Staubli VAL3: sendAckIO.pgx

public program sendAckIO(sio& x_sSocket, num& x_nConnFlag, RosSimpleMsg& x_rMsg, num& x_nMsgRecvState)
begin
  // Copyright (c) 2016, Ocado Technology - Robotics Research Team
  //
  // Licensed under the Apache License, Version 2.0 (the "License");
  // you may not use this file except in compliance with the License.
  // You may obtain a copy of the License at
  //
  //     http://www.apache.org/licenses/LICENSE-2.0
  //
  // Unless required by applicable law or agreed to in writing, software
  // distributed under the License is distributed on an "AS IS" BASIS,
  // WITHOUT WARRANTIES OR CONDITIONS OF ANY KIND, either express or implied.
  // See the License for the specific language governing permissions and
  // limitations under the License.



  switch x_rMsg.header.nMsgType
    case nStdMsgType["JOINT_TRAJ_PT"]
      call sendRosMsg(siTcpIpMotion, rosTrajPtAck.prefix, rosTrajPtAck.header, rosTrajPtAck.body, nInConnFlag)
    break
    case nStdMsgType["JOINT_TRAJ_PT_FULL"]
      call sendRosMsg(siTcpIpMotion, rosTrajPtFAck.prefix, rosTrajPtFAck.header, rosTrajPtFAck.body, nInConnFlag)
    break
    case Staubli:MsgType.WRITE_SINGLE_IO
      call sendRosMsg(x_sSocket, Staubli:writeSingIOAck.prefix, Staubli:writeSingIOAck.header, Staubli:writeSingIOAck.body, x_nConnFlag)
    break
    default
    break
  endSwitch

  // regardless of result from sending ACK
  // reset state machine to receive new messages
  x_nMsgRecvState=nReset
end
